FUNCTION_BLOCK FB_Transport_E
VAR_INPUT
	//Hardware Singale
	bSens1 :BOOL;
	bSens2 :BOOL;
	bSens3 :BOOL;
	bSens4 :BOOL;
END_VAR
VAR_OUTPUT
	bStation1 :BOOL;
	bStation2 :BOOL;
	bStation3 :BOOL;
	bStation4 :BOOL;
END_VAR
VAR
END_VAR

bStation1 :=bSens1;
bStation2 :=bSens2;
bStation3 :=bSens3;
bStation4 :=bSens4;

END_FUNCTION_BLOCK

(* stored: Version 1.1.0.1, ProductVersion 3.1.4024.15
   POU FB_Transport_E: Id {33754491-3b8e-48fa-8d65-817ba14d4b90}, SpecialFunc None *)
